FUNCTION_BLOCK FB_InterfaceSimulated IMPLEMENTS ITF_Cell
VAR_INPUT
END_VAR
VAR_OUTPUT
END_VAR
VAR
	 iTimer : INT;
	 iWaitingTime : INT := 500;
END_VAR

METHOD GetEmergencyOff : BOOL
VAR_INPUT
END_VAR

iTimer := iTimer +1;

IF iTimer > iWaitingTime THEN
	GetEmergencyOff := TRUE;
	iTimer := 0;	
END_IF
END_METHOD

METHOD GetEmergencyStop : BOOL
VAR_INPUT
END_VAR

iTimer := iTimer +1;

IF iTimer > iWaitingTime THEN
	GetEmergencyStop := TRUE;
	iTimer := 0;	
END_IF
END_METHOD

METHOD GetFinished : BOOL
VAR_INPUT
END_VAR

iTimer := iTimer +1;

IF iTimer > iWaitingTime THEN
	GetFinished := TRUE;
	iTimer := 0;	
END_IF
END_METHOD

METHOD GetIsRunning : BOOL
VAR_INPUT
END_VAR


iTimer := iTimer +1;

IF iTimer > iWaitingTime THEN
	GetIsRunning := TRUE;
	iTimer := 0;	
END_IF
END_METHOD

METHOD GetLoadPos : BOOL
VAR_INPUT
END_VAR


iTimer := iTimer +1;

IF iTimer > iWaitingTime THEN
	GetLoadPos := TRUE;
	iTimer := 0;	
END_IF
END_METHOD

METHOD GetStandby : BOOL
VAR_INPUT
END_VAR


iTimer := iTimer +1;

IF iTimer > iWaitingTime THEN
	GetStandby := TRUE;
	iTimer := 0;	
END_IF
END_METHOD

METHOD GetStartable : BOOL
VAR_INPUT
END_VAR



iTimer := iTimer +1;

IF iTimer > iWaitingTime THEN
	GetStartable := TRUE;
	iTimer := 0;	
END_IF
END_METHOD

METHOD GetUnloadPos : BOOL
VAR_INPUT
END_VAR


iTimer := iTimer +1;

IF iTimer > iWaitingTime THEN
	GetUnloadPos := TRUE;
	iTimer := 0;	
END_IF
END_METHOD

METHOD SetEmergencyOff : BOOL
VAR_INPUT
	b:BOOL;
END_VAR
END_METHOD

METHOD SetEmergencyStop : BOOL
VAR_INPUT
	b:BOOL;
END_VAR
END_METHOD

METHOD SetLoadPlace : BOOL
VAR_INPUT
	b :BOOL;
END_VAR
END_METHOD

METHOD SetMoveToLoad : BOOL
VAR_INPUT
	b:BOOL;
END_VAR
END_METHOD

METHOD SetMoveToUnload : BOOL
VAR_INPUT
	b:BOOL;
END_VAR
END_METHOD

METHOD SetStandby : BOOL
VAR_INPUT
	b:BOOL;
END_VAR
END_METHOD

METHOD SetStart : BOOL
VAR_INPUT
	b:BOOL;
END_VAR
END_METHOD

END_FUNCTION_BLOCK

(* stored: Version 1.1.0.1, ProductVersion 3.1.4024.0
   POU FB_InterfaceSimulated: Id {711cd097-7162-4d64-9799-f252f00dfb4a}, SpecialFunc None
   Method GetEmergencyOff: Id {a3778c58-2539-4411-a535-afc39b7e64b7}
   Method GetEmergencyStop: Id {4793d486-231e-46c0-b742-f27fe9a2dd46}
   Method GetFinished: Id {f0419497-82dc-4b93-90c9-165e09b123a2}
   Method GetIsRunning: Id {bd6844ff-30fb-40e6-83ea-047247412c2d}
   Method GetLoadPos: Id {a0995c13-d139-4bda-b1de-ab26cea30734}
   Method GetStandby: Id {d367178f-773e-4c12-8872-80e0b22f7231}
   Method GetStartable: Id {169a33e6-e097-4907-96ae-30e4eb031517}
   Method GetUnloadPos: Id {74d2db1f-c459-4bcd-885c-d3a0b624af62}
   Method SetEmergencyOff: Id {8e2e35d5-0985-4e0f-a33a-a1596c074c59}
   Method SetEmergencyStop: Id {05c98e4a-4181-4ae9-addd-e5c1df4fbdfc}
   Method SetLoadPlace: Id {f8bb8249-33db-4809-806d-7bfd2982bb05}
   Method SetMoveToLoad: Id {1606b5b0-686a-4313-8554-4dea48b0e96f}
   Method SetMoveToUnload: Id {87d7cc4c-8fa4-4a8c-a25b-fb7ca321ee18}
   Method SetStandby: Id {11266cf8-a5b9-46b4-8609-c4a888f97fc6}
   Method SetStart: Id {fb60e8a8-7fb5-4c12-881d-e417cce4b90d} *)
